SUBAPPLICATION ILOCK_SWITCH_2_QXA_OPC (* 2-Richtungs-Doppelwirkungs-Ausgang (Last-Wins mit Schutzzeit): je Richtung wird das echte Funktions-Kommando (Remote-Subscribe) mit dem bestehenden IO-Test-Kommando (Remote-Subscribe) per AX_OR_2 zusammengefuehrt, bevor es in den Interlock geht - IO-Test bleibt nutzbar, kann aber die beiden Richtungen nicht mehr dauerhaft gleichzeitig schalten. Interlocked Ausgang treibt den physischen logiBUS-Kanal UND meldet seinen tatsaechlichen Zustand sowohl an die bestehende IO-Test-Ueberwachung als auch an die echte Funktions-Rueckmeldung (z.B. GreenWhiteBackground am SoftKey) zurueck. Generisch fuer jeden 'digital DW'-Aktor (siehe IO-Liste_Vereinheitlicht.md) mit Bedienung von einem Modul ohne eigenes VT. *)
  (* Standard: 61499-2 *)
  (* Version 1.0, 2026-09-05, franz, Meisterschulen am Ostbahnhof *)
  PACKAGE MyLib::sys;
  IMPORT logiBUS::io::DQ::logiBUS_DO;
  IMPORT logiBUS::io::DQ::logiBUS_DO_S;
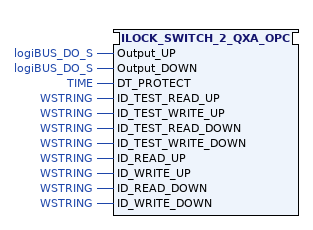
  VAR_INPUT
    Output_UP : logiBUS::io::DQ::logiBUS_DO_S := logiBUS_DO::Invalid; (* Physischer Ausgang Richtung UP/Links *)
    Output_DOWN : logiBUS::io::DQ::logiBUS_DO_S := logiBUS_DO::Invalid; (* Physischer Ausgang Richtung DOWN/Rechts *)
    DT_PROTECT : TIME := T#300ms; (* Schutz-Totzeit vor Richtungswechsel *)
    ID_TEST_READ_UP : WSTRING; (* Bestehende IO-Test-Subscribe-Adresse UP (z.B. STG3_Q0x_READ) *)
    ID_TEST_WRITE_UP : WSTRING; (* Bestehende IO-Test-Publish-Adresse UP (z.B. STG3_Q0x_WRITE) *)
    ID_TEST_READ_DOWN : WSTRING; (* Bestehende IO-Test-Subscribe-Adresse DOWN *)
    ID_TEST_WRITE_DOWN : WSTRING; (* Bestehende IO-Test-Publish-Adresse DOWN *)
    ID_READ_UP : WSTRING; (* Echtes Funktions-Kommando UP (Subscribe) *)
    ID_WRITE_UP : WSTRING; (* Echte Funktions-Rueckmeldung UP (Publish) *)
    ID_READ_DOWN : WSTRING; (* Echtes Funktions-Kommando DOWN (Subscribe) *)
    ID_WRITE_DOWN : WSTRING; (* Echte Funktions-Rueckmeldung DOWN (Publish) *)
  END_VAR
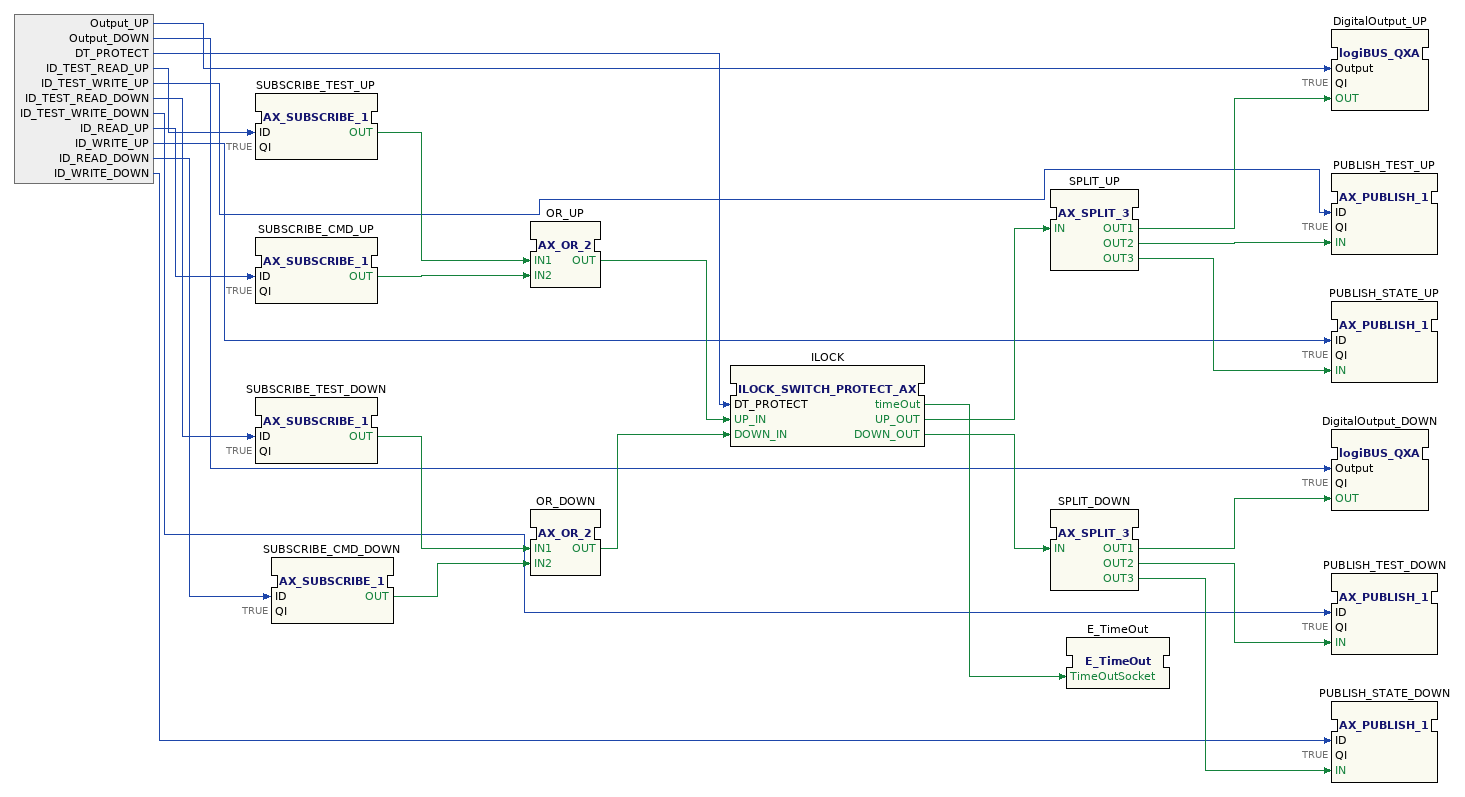
  FBS
    SUBSCRIBE_TEST_UP : adapter::net::AX_SUBSCRIBE_1(QI := TRUE);
    SUBSCRIBE_CMD_UP : adapter::net::AX_SUBSCRIBE_1(QI := TRUE);
    OR_UP : adapter::booleanOperators::AX_OR_2;
    SUBSCRIBE_TEST_DOWN : adapter::net::AX_SUBSCRIBE_1(QI := TRUE);
    SUBSCRIBE_CMD_DOWN : adapter::net::AX_SUBSCRIBE_1(QI := TRUE);
    OR_DOWN : adapter::booleanOperators::AX_OR_2;
    ILOCK : logiBUS::signalprocessing::interlock::ILOCK_SWITCH_PROTECT_AX;
    E_TimeOut : iec61499::events::E_TimeOut;
    SPLIT_UP : adapter::events::unidirectional::AX_SPLIT_3;
    SPLIT_DOWN : adapter::events::unidirectional::AX_SPLIT_3;
    DigitalOutput_UP : logiBUS::io::DQ::logiBUS_QXA(QI := TRUE);
    DigitalOutput_DOWN : logiBUS::io::DQ::logiBUS_QXA(QI := TRUE);
    PUBLISH_TEST_UP : adapter::net::AX_PUBLISH_1(QI := TRUE);
    PUBLISH_STATE_UP : adapter::net::AX_PUBLISH_1(QI := TRUE);
    PUBLISH_TEST_DOWN : adapter::net::AX_PUBLISH_1(QI := TRUE);
    PUBLISH_STATE_DOWN : adapter::net::AX_PUBLISH_1(QI := TRUE);
  END_FBS
  DATA_CONNECTIONS
    ID_TEST_READ_UP TO SUBSCRIBE_TEST_UP.ID;
    ID_READ_UP TO SUBSCRIBE_CMD_UP.ID;
    ID_TEST_READ_DOWN TO SUBSCRIBE_TEST_DOWN.ID;
    ID_READ_DOWN TO SUBSCRIBE_CMD_DOWN.ID;
    DT_PROTECT TO ILOCK.DT_PROTECT;
    Output_UP TO DigitalOutput_UP.Output;
    Output_DOWN TO DigitalOutput_DOWN.Output;
    ID_TEST_WRITE_UP TO PUBLISH_TEST_UP.ID;
    ID_WRITE_UP TO PUBLISH_STATE_UP.ID;
    ID_TEST_WRITE_DOWN TO PUBLISH_TEST_DOWN.ID;
    ID_WRITE_DOWN TO PUBLISH_STATE_DOWN.ID;
  END_CONNECTIONS
  ADAPTER_CONNECTIONS
    SUBSCRIBE_TEST_UP.OUT TO OR_UP.IN1;
    SUBSCRIBE_CMD_UP.OUT TO OR_UP.IN2;
    OR_UP.OUT TO ILOCK.UP_IN;
    SUBSCRIBE_TEST_DOWN.OUT TO OR_DOWN.IN1;
    SUBSCRIBE_CMD_DOWN.OUT TO OR_DOWN.IN2;
    OR_DOWN.OUT TO ILOCK.DOWN_IN;
    ILOCK.timeOut TO E_TimeOut.TimeOutSocket;
    ILOCK.UP_OUT TO SPLIT_UP.IN;
    SPLIT_UP.OUT1 TO DigitalOutput_UP.OUT;
    SPLIT_UP.OUT2 TO PUBLISH_TEST_UP.IN;
    SPLIT_UP.OUT3 TO PUBLISH_STATE_UP.IN;
    ILOCK.DOWN_OUT TO SPLIT_DOWN.IN;
    SPLIT_DOWN.OUT1 TO DigitalOutput_DOWN.OUT;
    SPLIT_DOWN.OUT2 TO PUBLISH_TEST_DOWN.IN;
    SPLIT_DOWN.OUT3 TO PUBLISH_STATE_DOWN.IN;
  END_CONNECTIONS
END_SUBAPPLICATION
